{attribute 'qualified_only'}
VAR_GLOBAL
	{attribute 'TcInitSymbol'}
	sTcpHost   : STRING(15) := '127.0.0.1';
	{attribute 'TcInitSymbol'}
	nTcpPort   : UINT := 502;
	{attribute 'TcInitSymbol'}
	nDemoUnit  : USINT := 1;
	{attribute 'TcInitSymbol'}
	nMeterUnit : USINT := 1;
END_VAR

(* stored: Version 1.1.0.1
   GVL GVL_Site: Id {40ca1e0d-e09c-41ca-b674-bc1f196f7d3d} *)
